(* Logix 5000 project; controller Close_Palletizing 1769-L33ERM rev 33.13; software revision 33.00; part 3 of 5 *)

ADD_ON_INSTRUCTION Generic_4PORT_IOL   (* revision 2.0 *)
// Revision note:
// 4/7/20: Changed the Input values to an input array. This makes copying the information more usable and also allows for the full Port_Process_Data_Size length.
VAR_OUTPUT
   IOL_Mode : BOOL; {access Read Only, visible}
END_VAR
VAR_IN_OUT
   PLC_Input : INT[123]; {required}
   PLC_Output : INT[87]; {required}
END_VAR
VAR_INPUT
   Port_Process_Data_Size : INT := 4; {visible}
   Port_Number : INT; {visible}
END_VAR
VAR_OUTPUT
   Vendor_ID : INT; {access Read Only, visible}
   Device_ID : DINT; {access Read Only, visible}
END_VAR
VAR_IN_OUT
   Input_Data_Array : INT[16]; {required}
   Output_Data_Array : INT[16]; {required}
END_VAR
VAR_OUTPUT
   Device_Not_Connected : BOOL; {access Read Only, visible}
   Invalid_Data : BOOL; {access Read Only, visible}
   Wrong_VID_DID : BOOL; {access Read Only, visible}
   AOI_Settings_Error : BOOL; {access Read Only, visible}
END_VAR
VAR
   Data_Size : INT; {access None}
   Offset_Address : INT; {access None}
   Offset_StatusFlgs : INT; {access None}
   Process_Offset : INT; {access None}
   RealPort_Num : INT; {access None}
   StatusFlgs_Offset : INT; {access None}
   Process_Out_Offset : INT; {access None}
END_VAR

ROUTINE Logic   (* ladder *)
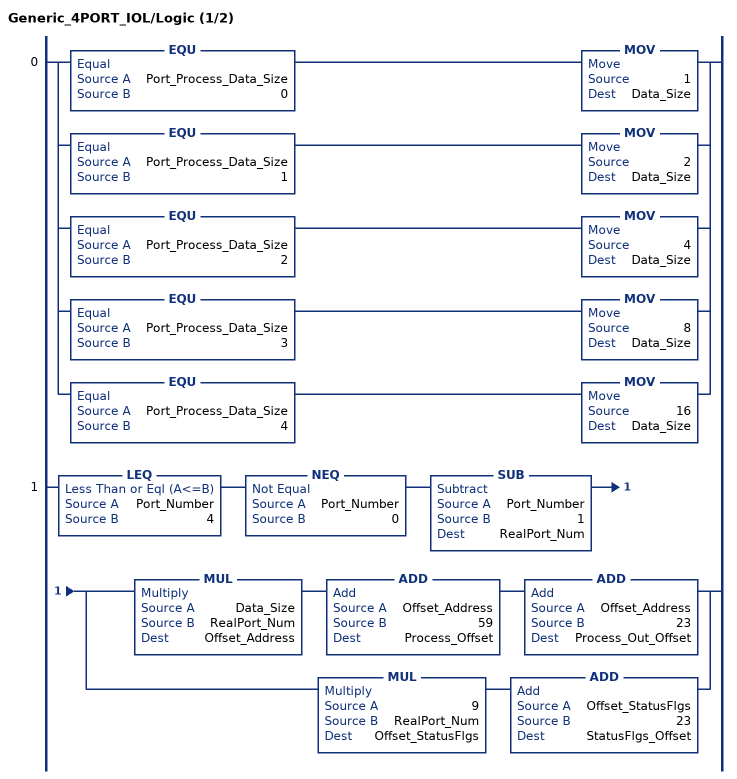
   0: [EQU(Port_Process_Data_Size,0) MOV(1,Data_Size) ,EQU(Port_Process_Data_Size,1) MOV(2,Data_Size) ,EQU(Port_Process_Data_Size,2) MOV(4,Data_Size) ,EQU(Port_Process_Data_Size,3) MOV(8,Data_Size) ,EQU(Port_Process_Data_Size,4) MOV(16,Data_Size) ];
   1: LEQ(Port_Number,4)NEQ(Port_Number,0)SUB(Port_Number,1,RealPort_Num)[MUL(Data_Size,RealPort_Num,Offset_Address) ADD(Offset_Address,59,Process_Offset) ADD(Offset_Address,23,Process_Out_Offset) ,MUL(9,RealPort_Num,Offset_StatusFlgs) ADD(Offset_StatusFlgs,23,StatusFlgs_Offset) ];
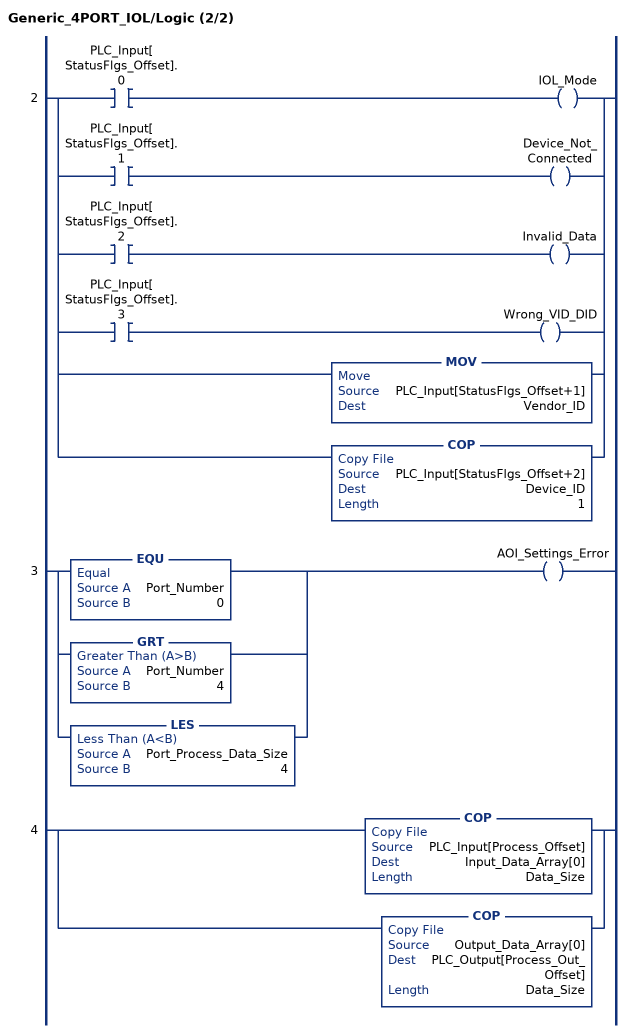
   2: [XIC(PLC_Input[StatusFlgs_Offset].0) OTE(IOL_Mode) ,XIC(PLC_Input[StatusFlgs_Offset].1) OTE(Device_Not_Connected) ,XIC(PLC_Input[StatusFlgs_Offset].2) OTE(Invalid_Data) ,XIC(PLC_Input[StatusFlgs_Offset].3) OTE(Wrong_VID_DID) ,MOV(PLC_Input[StatusFlgs_Offset+1],Vendor_ID) ,COP(PLC_Input[StatusFlgs_Offset+2],Device_ID,1) ];
   3: [EQU(Port_Number,0) ,GRT(Port_Number,4) ,LES(Port_Process_Data_Size,4) ]OTE(AOI_Settings_Error);
   4: [COP(PLC_Input[Process_Offset],Input_Data_Array[0],Data_Size) ,COP(Output_Data_Array[0],PLC_Output[Process_Out_Offset],Data_Size) ];
END_ROUTINE
END_ADD_ON_INSTRUCTION

ADD_ON_INSTRUCTION LMT_4PORT_IOL   (* revision 1.0, vendor ifm efector *)
// Cyclic Data with Diagnostics
// Revision note:
// 07/08/19 - HT
VAR_IN_OUT
   PLC_Input : INT[123]; {required}
END_VAR
VAR_INPUT
   Port_Process_Data_Size : INT := 4; {visible}
   Port_Number : INT; {visible}
END_VAR
VAR_OUTPUT
   Datastorage_Error : BOOL; {access Read Only, visible}
   Process_Data : INT; {access Read Only}
   Device_Not_Connected : BOOL; {access Read Only, visible}
   IOL_Mode : BOOL; {access Read Only, visible}
   Invalid_Data : BOOL; {access Read Only, visible}
   Media_Value : INT; {access Read Only, visible}
   Wrong_VID_DID : BOOL; {access Read Only, visible}
   Out1 : BOOL; {access Read Only, visible}
   Vendor_ID : INT; {access Read Only, visible}
   Device_ID : INT; {access Read Only, visible}
   Out2 : BOOL; {access Read Only, visible}
END_VAR
VAR
   RealPort_Num : INT; {access None}
   Offset_Address : INT; {access None}
   Process_PDI : INT; {access None}
   Process_Offset : INT; {access None}
   Offset_StatusFlgs : INT; {access None}
   StatusFlgs_Offset : INT; {access None}
   Data_Size : INT; {access None}
   Pressure_msk : INT; {access None}
END_VAR

ROUTINE Logic   (* ladder *)
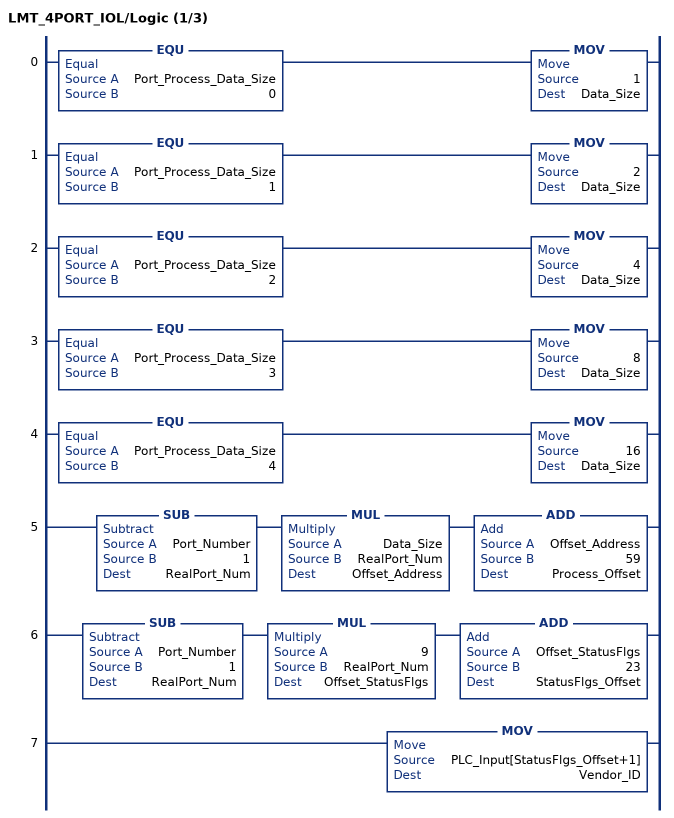
   0: EQU(Port_Process_Data_Size,0)MOV(1,Data_Size);
   1: EQU(Port_Process_Data_Size,1)MOV(2,Data_Size);
   2: EQU(Port_Process_Data_Size,2)MOV(4,Data_Size);
   3: EQU(Port_Process_Data_Size,3)MOV(8,Data_Size);
   4: EQU(Port_Process_Data_Size,4)MOV(16,Data_Size);
   5: SUB(Port_Number,1,RealPort_Num)MUL(Data_Size,RealPort_Num,Offset_Address)ADD(Offset_Address,59,Process_Offset);
   6: SUB(Port_Number,1,RealPort_Num)MUL(9,RealPort_Num,Offset_StatusFlgs)ADD(Offset_StatusFlgs,23,StatusFlgs_Offset);
   7: MOV(PLC_Input[StatusFlgs_Offset+1],Vendor_ID);
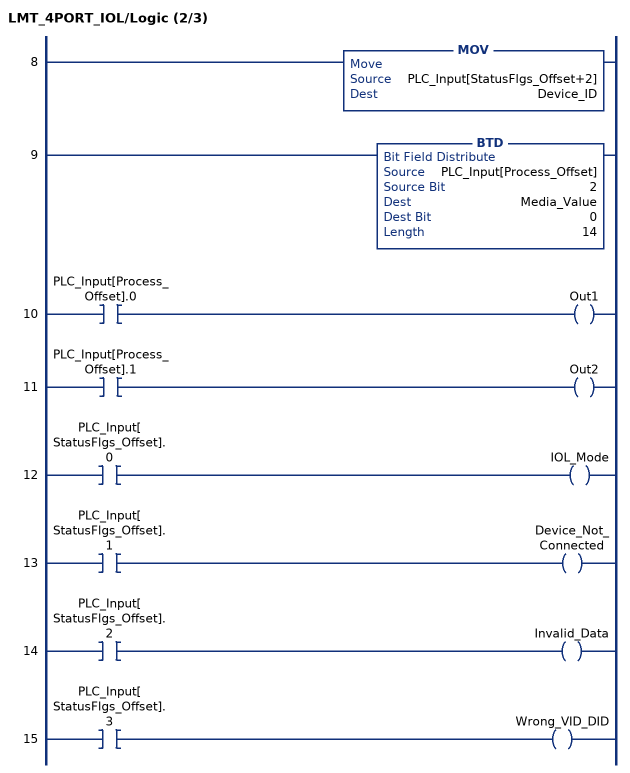
   8: MOV(PLC_Input[StatusFlgs_Offset+2],Device_ID);
   9: BTD(PLC_Input[Process_Offset],2,Media_Value,0,14);
   10: XIC(PLC_Input[Process_Offset].0)OTE(Out1);
   11: XIC(PLC_Input[Process_Offset].1)OTE(Out2);
   12: XIC(PLC_Input[StatusFlgs_Offset].0)OTE(IOL_Mode);
   13: XIC(PLC_Input[StatusFlgs_Offset].1)OTE(Device_Not_Connected);
   14: XIC(PLC_Input[StatusFlgs_Offset].2)OTE(Invalid_Data);
   15: XIC(PLC_Input[StatusFlgs_Offset].3)OTE(Wrong_VID_DID);
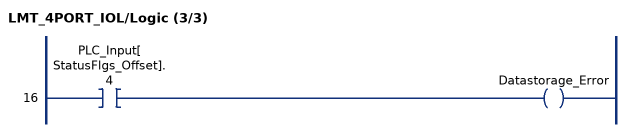
   16: XIC(PLC_Input[StatusFlgs_Offset].4)OTE(Datastorage_Error);
END_ROUTINE
END_ADD_ON_INSTRUCTION

ADD_ON_INSTRUCTION LT_4PORT_IOL   (* revision 1.0, vendor ifm efector *)
// Cyclic Data with Diagnostics
// Revision note:
// 07/08/19 - HT
VAR_IN_OUT
   PLC_Input : INT[123]; {required}
END_VAR
VAR_INPUT
   Port_Process_Data_Size : INT := 4; {visible}
   Port_Number : INT; {visible}
   Temp_Value_Gradient : REAL := 0.1; {visible}
   Level_Value_Gradient : REAL := 0.1; {visible}
END_VAR
VAR_OUTPUT
   Temperature : REAL; {access Read Only, visible}
   Datastorage_Error : BOOL; {access Read Only, visible}
   Process_Data : INT; {access Read Only}
   Device_Not_Connected : BOOL; {access Read Only, visible}
   IOL_Mode : BOOL; {access Read Only, visible}
   Invalid_Data : BOOL; {access Read Only, visible}
   Wrong_VID_DID : BOOL; {access Read Only, visible}
   Level : REAL; {access Read Only, visible}
   Out1 : BOOL; {access Read Only, visible}
   Out2 : BOOL; {access Read Only, visible}
   Vendor_ID : INT; {access Read Only, visible}
   Device_ID : INT; {access Read Only, visible}
   Out3 : BOOL; {access Read Only, visible}
   Out4 : BOOL; {access Read Only, visible}
END_VAR
VAR
   RealPort_Num : INT; {access None}
   Offset_Address : INT; {access None}
   Process_PDI : INT; {access None}
   Process_Offset : INT; {access None}
   Offset_StatusFlgs : INT; {access None}
   StatusFlgs_Offset : INT; {access None}
   Data_Size : INT; {access None}
END_VAR

ROUTINE Logic   (* ladder *)
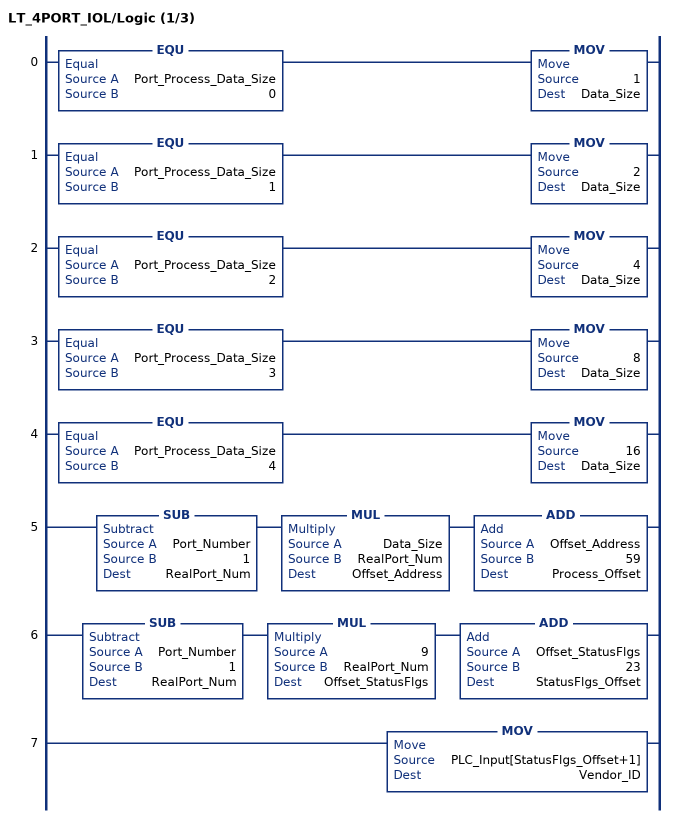
   0: EQU(Port_Process_Data_Size,0)MOV(1,Data_Size);
   1: EQU(Port_Process_Data_Size,1)MOV(2,Data_Size);
   2: EQU(Port_Process_Data_Size,2)MOV(4,Data_Size);
   3: EQU(Port_Process_Data_Size,3)MOV(8,Data_Size);
   4: EQU(Port_Process_Data_Size,4)MOV(16,Data_Size);
   5: SUB(Port_Number,1,RealPort_Num)MUL(Data_Size,RealPort_Num,Offset_Address)ADD(Offset_Address,59,Process_Offset);
   6: SUB(Port_Number,1,RealPort_Num)MUL(9,RealPort_Num,Offset_StatusFlgs)ADD(Offset_StatusFlgs,23,StatusFlgs_Offset);
   7: MOV(PLC_Input[StatusFlgs_Offset+1],Vendor_ID);
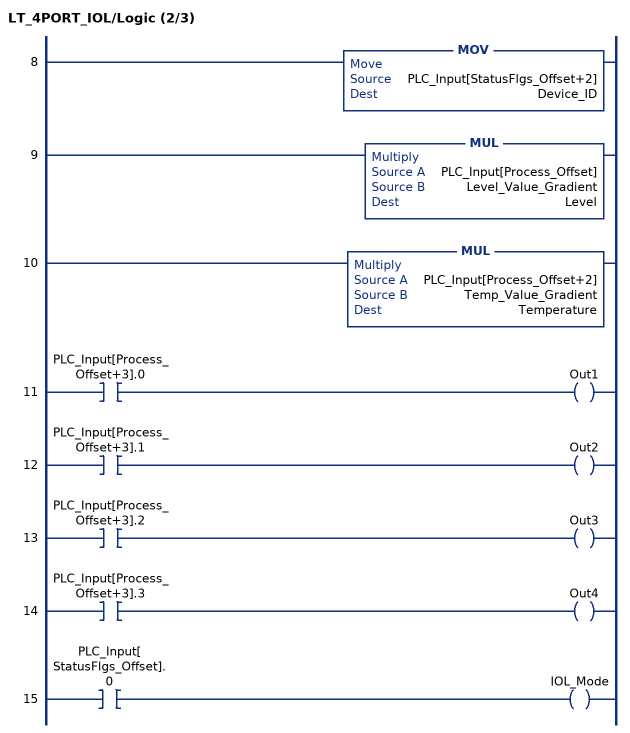
   8: MOV(PLC_Input[StatusFlgs_Offset+2],Device_ID);
   9: MUL(PLC_Input[Process_Offset],Level_Value_Gradient,Level);
   10: MUL(PLC_Input[Process_Offset+2],Temp_Value_Gradient,Temperature);
   11: XIC(PLC_Input[Process_Offset+3].0)OTE(Out1);
   12: XIC(PLC_Input[Process_Offset+3].1)OTE(Out2);
   13: XIC(PLC_Input[Process_Offset+3].2)OTE(Out3);
   14: XIC(PLC_Input[Process_Offset+3].3)OTE(Out4);
   15: XIC(PLC_Input[StatusFlgs_Offset].0)OTE(IOL_Mode);
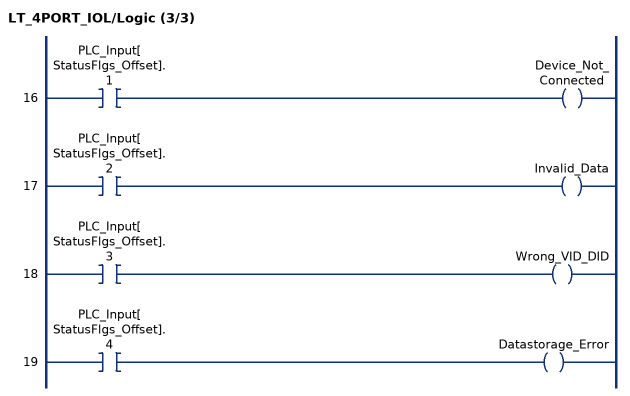
   16: XIC(PLC_Input[StatusFlgs_Offset].1)OTE(Device_Not_Connected);
   17: XIC(PLC_Input[StatusFlgs_Offset].2)OTE(Invalid_Data);
   18: XIC(PLC_Input[StatusFlgs_Offset].3)OTE(Wrong_VID_DID);
   19: XIC(PLC_Input[StatusFlgs_Offset].4)OTE(Datastorage_Error);
END_ROUTINE
END_ADD_ON_INSTRUCTION

ADD_ON_INSTRUCTION Two_AcyclicCmds_4P   (* revision 1.1 *)
// Revision note:
// 3/26/20 : On device not connected the Cmd1_DN, Cmd2_DN, Cmds_DN and Cmd_Error output bits are unlatched.
// If all Cmd Index 0, then commands are still cycled so the AL1x2x_Rdy an Cmds_DN bit still toggle on/off when the AOI is triggered.
VAR_IN_OUT
   PLC_Input : INT[123]; {required}
   PLC_Output : INT[87]; {required}
END_VAR
VAR_OUTPUT
   IOL_Mode : BOOL; {visible}
   Device_Not_Connected : BOOL; {access Read Only, visible}
   AL1x2x_Cmd_Rdy : BOOL; {visible}
   AOI_Settings_Error : BOOL; {visible}
   Cmds_Busy : BOOL; {visible}
   Cmd1_DN : BOOL; {visible}
   Cmd2_DN : BOOL; {visible}
   Cmds_DN : BOOL; {visible}
   Cmd_Errors : BOOL; {visible}
END_VAR
VAR_IN_OUT
   IOLinkMaster_Name : DINT; {required}
END_VAR
VAR_INPUT
   Port_Number : SINT; {visible}
END_VAR
VAR_OUTPUT
   Vendor_ID : INT; {access Read Only, visible}
   Device_ID : INT; {access Read Only, visible}
END_VAR
VAR_INPUT
   Cmd1_Index : INT; {visible}
   Cmd1_Subindex : INT; {visible}
   Cmd1_Rd_Wr : SINT; {visible}
   Cmd1_ByteLength : SINT; {visible}
END_VAR
VAR_IN_OUT
   Cmd1_RdWr_Buffer : SINT[32]; {required}
END_VAR
VAR_INPUT
   Cmd2_Index : INT; {visible}
   Cmd2_Subindex : INT; {visible}
   Cmd2_Rd_Wr : SINT; {visible}
   Cmd2_ByteLength : SINT; {visible}
END_VAR
VAR_IN_OUT
   Cmd2_RdWr_Buffer : SINT[32]; {required}
END_VAR
VAR_INPUT
   Cmd_Trigger : BOOL; {visible}
END_VAR
VAR_IN_OUT
   Cmd_Error_Codes : INT[2]; {required}
END_VAR
VAR_OUTPUT
   TimeOut : BOOL;
END_VAR
VAR
   Cmd1 : BOOL; {access None}
   Skip_Cmd1 : BOOL; {access None}
   Cmd1_DN_Error : BOOL; {access None}
   Cmd2 : BOOL; {access None}
   Skip_Cmd2 : BOOL; {access None}
   Cmd2_DN_Error : BOOL; {access None}
   Cmd1_Trigger : BOOL; {access None}
   Cmd2_Trigger : BOOL; {access None}
   Cmd1ReleaseTrigger : BOOL; {access None}
   Cmd2ReleaseTrigger : BOOL; {access None}
   Cmd2TriggerDelay : TIMER := (PRE := 20); {access None}
   Cmd1_PLC_OutTrigger : BOOL; {access None}
   TriggerCmdBuffer_ONS : BOOL; {access None}
   PLCTrigger : SINT; {access None}
   RealPort_Num : SINT; {access None}
   Offset_Address : INT; {access None}
   Cmd1_Busy : BOOL; {access None}
   Cmd2_Busy : BOOL; {access None}
   Offset_StatusFlgs : INT; {access None}
   StatusFlgs_Offset : INT; {access None}
   TimeOut1 : TIMER := (PRE := 6000); {access None}
   TimeOut2 : TIMER := (PRE := 6000); {access None}
   TimeOut1_Signal : BOOL; {access None}
   TimeOut2_Signal : BOOL; {access None}
   AL1x2x_Cmd_Rdy_Timer : TIMER := (PRE := 20); {access None}
   DevNotConn_Signal : BOOL; {access None}   // Signal to Latch when device is disconnected
   NoCmdSet : BOOL; {access None}
   SimCmdTimer : TIMER := (PRE := 20); {access None}
   Cmd2ReleaseTrigger_Signal : BOOL; {access None}
END_VAR

ROUTINE Logic   (* ladder *)
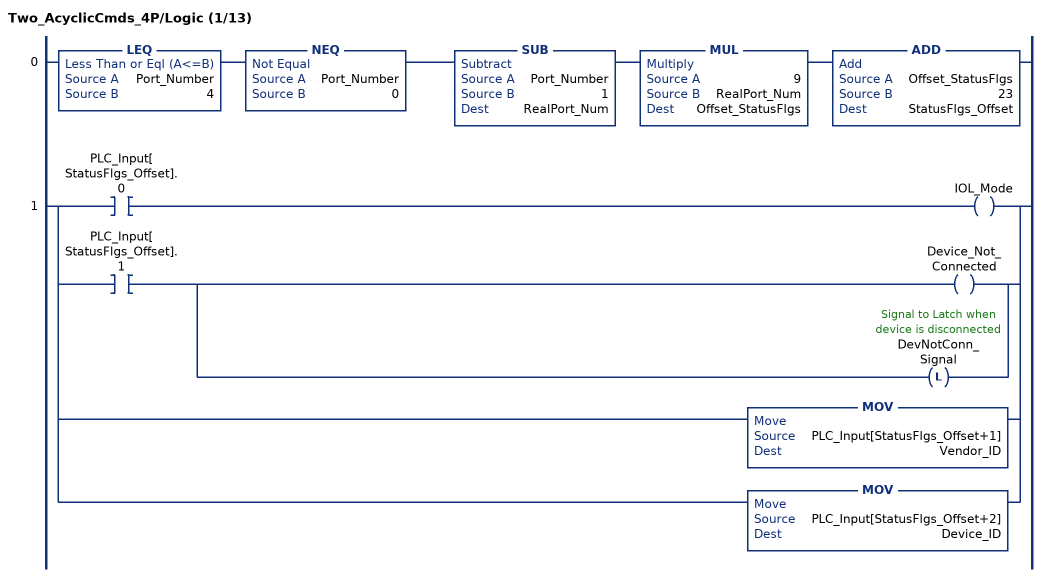
   0: LEQ(Port_Number,4)NEQ(Port_Number,0)SUB(Port_Number,1,RealPort_Num)MUL(9,RealPort_Num,Offset_StatusFlgs)ADD(Offset_StatusFlgs,23,StatusFlgs_Offset);
   1: [XIC(PLC_Input[StatusFlgs_Offset].0) OTE(IOL_Mode) ,XIC(PLC_Input[StatusFlgs_Offset].1) [OTE(Device_Not_Connected) ,OTL(DevNotConn_Signal) ] ,MOV(PLC_Input[StatusFlgs_Offset+1],Vendor_ID) ,MOV(PLC_Input[StatusFlgs_Offset+2],Device_ID) ];
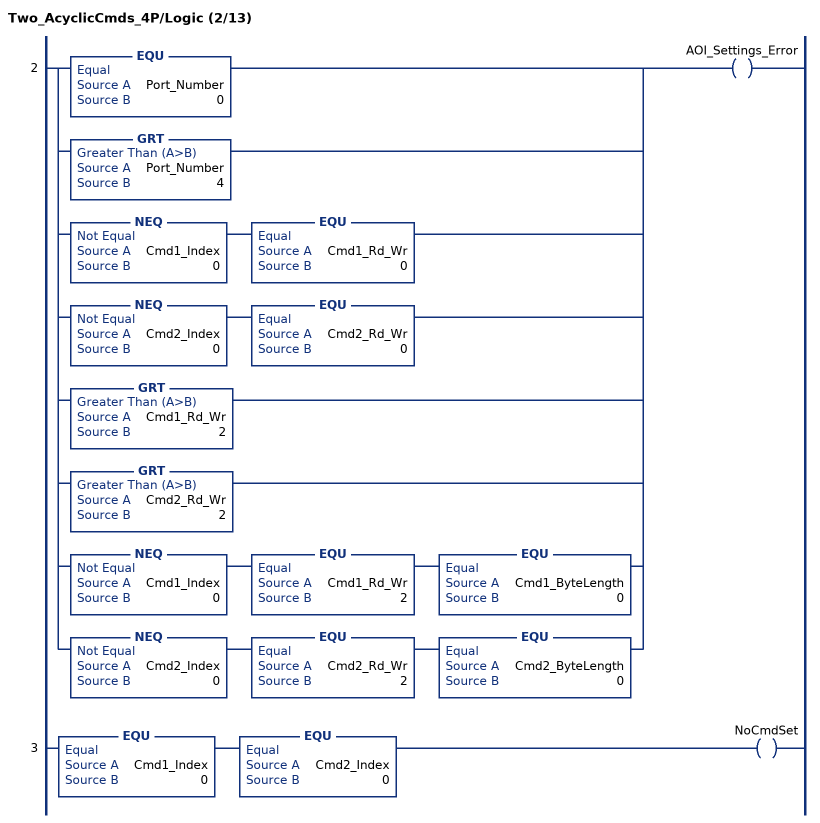
   2: [EQU(Port_Number,0) ,GRT(Port_Number,4) ,NEQ(Cmd1_Index,0) EQU(Cmd1_Rd_Wr,0) ,NEQ(Cmd2_Index,0) EQU(Cmd2_Rd_Wr,0) ,GRT(Cmd1_Rd_Wr,2) ,GRT(Cmd2_Rd_Wr,2) ,NEQ(Cmd1_Index,0) EQU(Cmd1_Rd_Wr,2) EQU(Cmd1_ByteLength,0) ,NEQ(Cmd2_Index,0) EQU(Cmd2_Rd_Wr,2) EQU(Cmd2_ByteLength,0) ]OTE(AOI_Settings_Error);
   3: EQU(Cmd1_Index,0)EQU(Cmd2_Index,0)OTE(NoCmdSet);
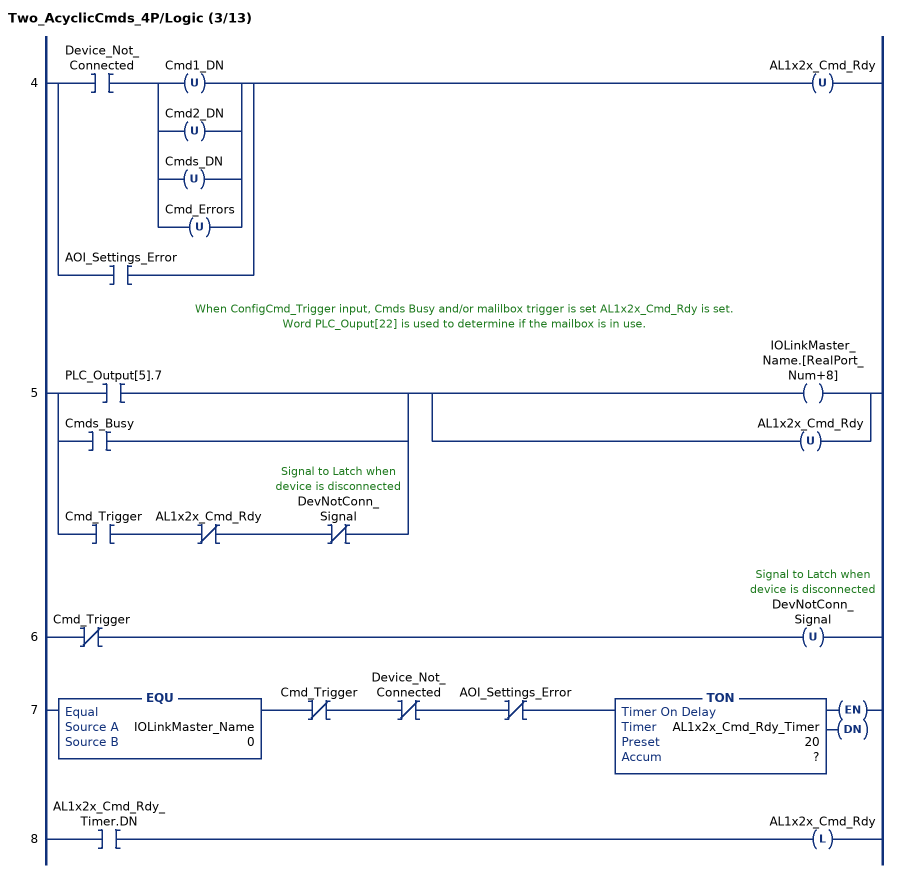
   4: [XIC(Device_Not_Connected) [OTU(Cmd1_DN) ,OTU(Cmd2_DN) ,OTU(Cmds_DN) ,OTU(Cmd_Errors) ] ,XIC(AOI_Settings_Error) ]OTU(AL1x2x_Cmd_Rdy);
   // When ConfigCmd_Trigger input, Cmds Busy and/or malilbox trigger is set AL1x2x_Cmd_Rdy is set.
   // Word PLC_Ouput[22] is used to determine if the mailbox is in use.
   5: [XIC(PLC_Output[5].7) ,XIC(Cmds_Busy) ,XIC(Cmd_Trigger) XIO(AL1x2x_Cmd_Rdy) XIO(DevNotConn_Signal) ][OTE(IOLinkMaster_Name.[RealPort_Num+8]) ,OTU(AL1x2x_Cmd_Rdy) ];
   6: XIO(Cmd_Trigger)OTU(DevNotConn_Signal);
   7: EQU(IOLinkMaster_Name,0)XIO(Cmd_Trigger)XIO(Device_Not_Connected)XIO(AOI_Settings_Error)TON(AL1x2x_Cmd_Rdy_Timer,?,?);
   8: XIC(AL1x2x_Cmd_Rdy_Timer.DN)OTL(AL1x2x_Cmd_Rdy);
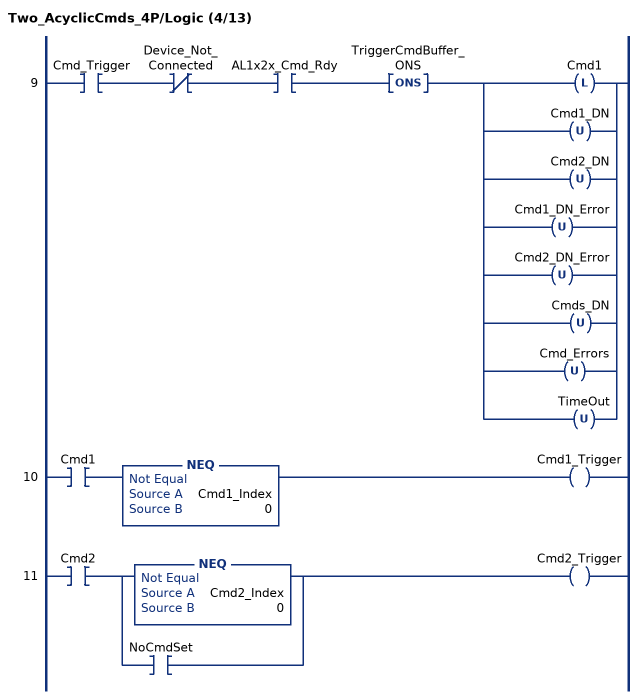
   9: XIC(Cmd_Trigger)XIO(Device_Not_Connected)XIC(AL1x2x_Cmd_Rdy)ONS(TriggerCmdBuffer_ONS)[OTL(Cmd1) ,[OTU(Cmd1_DN) ,OTU(Cmd2_DN) ,OTU(Cmd1_DN_Error) ,OTU(Cmd2_DN_Error) ,OTU(Cmds_DN) ,OTU(Cmd_Errors) ,OTU(TimeOut) ] ];
   10: XIC(Cmd1)NEQ(Cmd1_Index,0)OTE(Cmd1_Trigger);
   11: XIC(Cmd2)[NEQ(Cmd2_Index,0) ,XIC(NoCmdSet) ]OTE(Cmd2_Trigger);
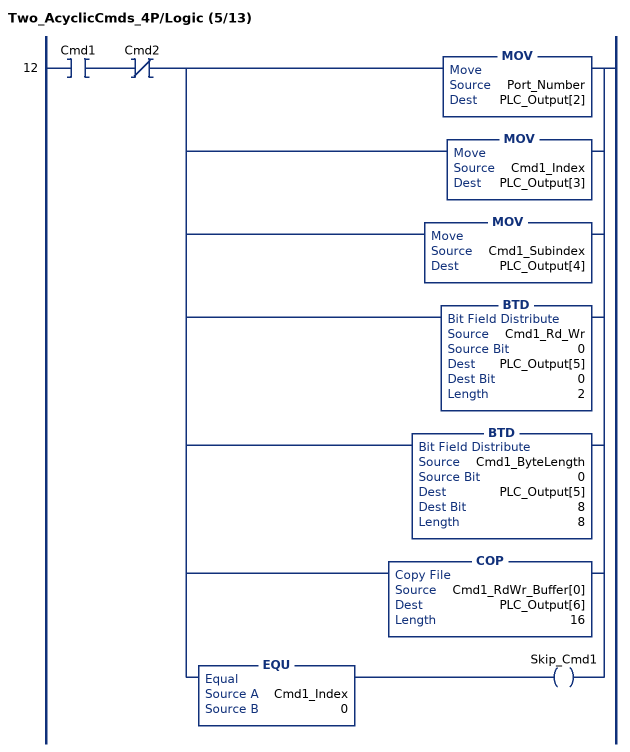
   12: XIC(Cmd1)XIO(Cmd2)[[MOV(Port_Number,PLC_Output[2]) ,MOV(Cmd1_Index,PLC_Output[3]) ,MOV(Cmd1_Subindex,PLC_Output[4]) ,BTD(Cmd1_Rd_Wr,0,PLC_Output[5],0,2) ,BTD(Cmd1_ByteLength,0,PLC_Output[5],8,8) ,COP(Cmd1_RdWr_Buffer[0],PLC_Output[6],16) ] ,EQU(Cmd1_Index,0) OTE(Skip_Cmd1) ];
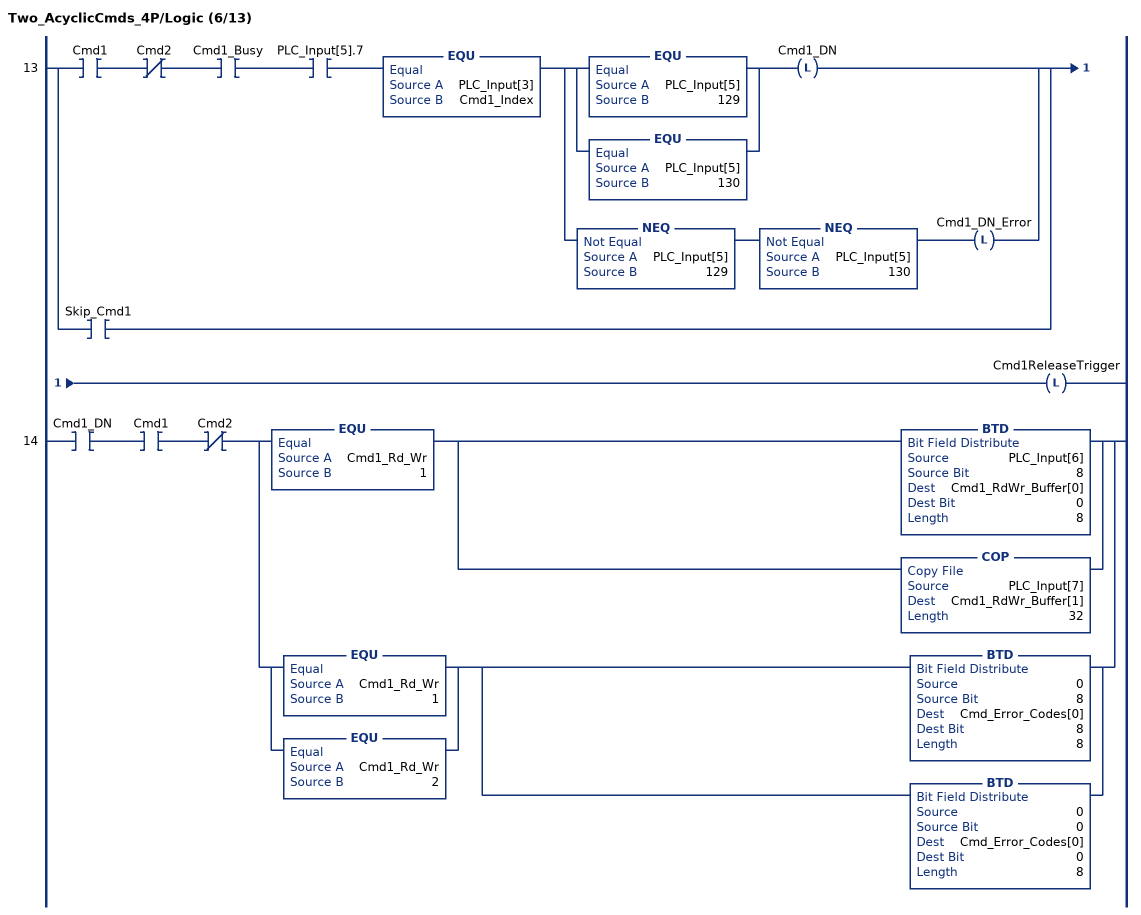
   13: [XIC(Cmd1) XIO(Cmd2) XIC(Cmd1_Busy) XIC(PLC_Input[5].7) EQU(PLC_Input[3],Cmd1_Index) [[EQU(PLC_Input[5],129) ,EQU(PLC_Input[5],130) ] OTL(Cmd1_DN) ,NEQ(PLC_Input[5],129) NEQ(PLC_Input[5],130) OTL(Cmd1_DN_Error) ] ,XIC(Skip_Cmd1) ]OTL(Cmd1ReleaseTrigger);
   14: XIC(Cmd1_DN)XIC(Cmd1)XIO(Cmd2)[EQU(Cmd1_Rd_Wr,1) [BTD(PLC_Input[6],8,Cmd1_RdWr_Buffer[0],0,8) ,COP(PLC_Input[7],Cmd1_RdWr_Buffer[1],32) ] ,[EQU(Cmd1_Rd_Wr,1) ,EQU(Cmd1_Rd_Wr,2) ] [BTD(0,8,Cmd_Error_Codes[0],8,8) ,BTD(0,0,Cmd_Error_Codes[0],0,8) ] ];
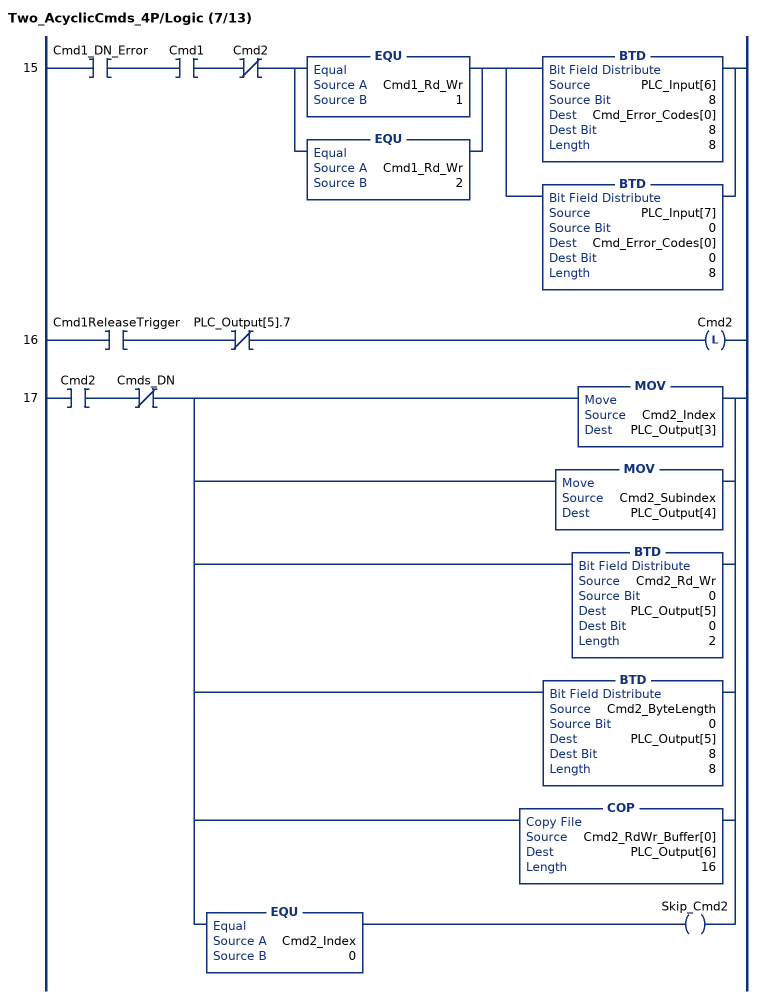
   15: XIC(Cmd1_DN_Error)XIC(Cmd1)XIO(Cmd2)[EQU(Cmd1_Rd_Wr,1) ,EQU(Cmd1_Rd_Wr,2) ][BTD(PLC_Input[6],8,Cmd_Error_Codes[0],8,8) ,BTD(PLC_Input[7],0,Cmd_Error_Codes[0],0,8) ];
   16: XIC(Cmd1ReleaseTrigger)XIO(PLC_Output[5].7)OTL(Cmd2);
   17: XIC(Cmd2)XIO(Cmds_DN)[[MOV(Cmd2_Index,PLC_Output[3]) ,MOV(Cmd2_Subindex,PLC_Output[4]) ,BTD(Cmd2_Rd_Wr,0,PLC_Output[5],0,2) ,BTD(Cmd2_ByteLength,0,PLC_Output[5],8,8) ,COP(Cmd2_RdWr_Buffer[0],PLC_Output[6],16) ] ,EQU(Cmd2_Index,0) OTE(Skip_Cmd2) ];
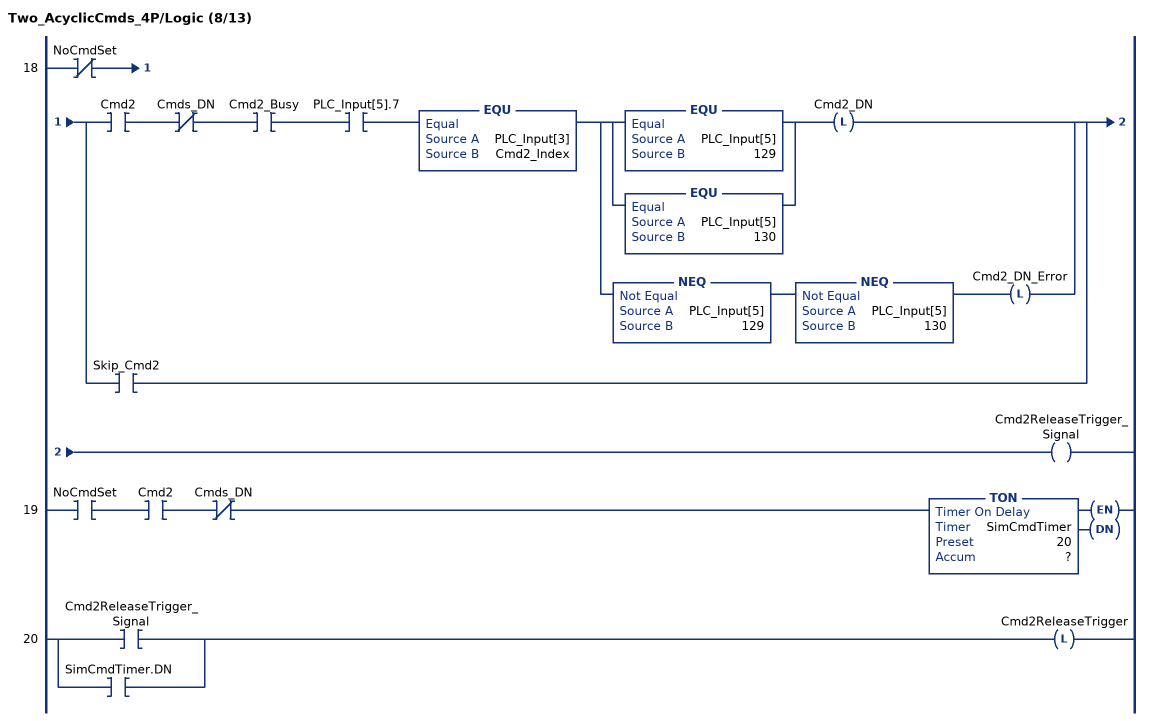
   18: XIO(NoCmdSet)[XIC(Cmd2) XIO(Cmds_DN) XIC(Cmd2_Busy) XIC(PLC_Input[5].7) EQU(PLC_Input[3],Cmd2_Index) [[EQU(PLC_Input[5],129) ,EQU(PLC_Input[5],130) ] OTL(Cmd2_DN) ,NEQ(PLC_Input[5],129) NEQ(PLC_Input[5],130) OTL(Cmd2_DN_Error) ] ,XIC(Skip_Cmd2) ]OTE(Cmd2ReleaseTrigger_Signal);
   19: XIC(NoCmdSet)XIC(Cmd2)XIO(Cmds_DN)TON(SimCmdTimer,?,?);
   20: [XIC(Cmd2ReleaseTrigger_Signal) ,XIC(SimCmdTimer.DN) ]OTL(Cmd2ReleaseTrigger);
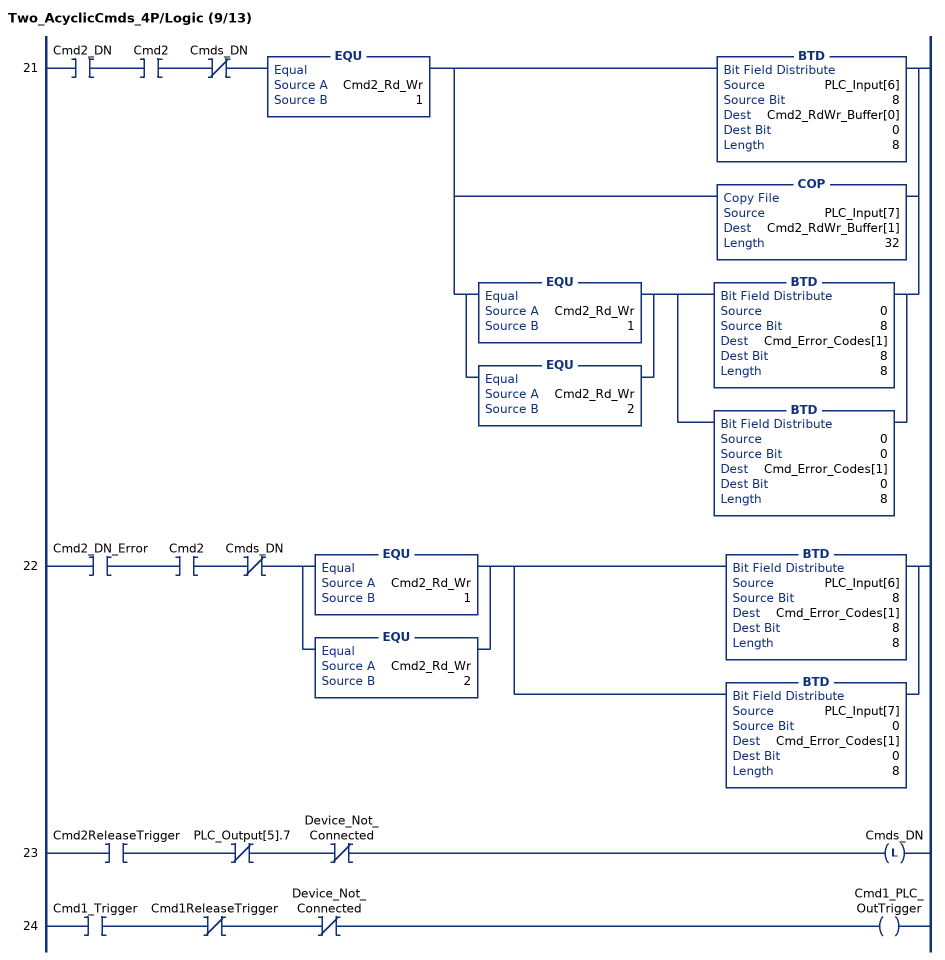
   21: XIC(Cmd2_DN)XIC(Cmd2)XIO(Cmds_DN)EQU(Cmd2_Rd_Wr,1)[[BTD(PLC_Input[6],8,Cmd2_RdWr_Buffer[0],0,8) ,COP(PLC_Input[7],Cmd2_RdWr_Buffer[1],32) ] ,[EQU(Cmd2_Rd_Wr,1) ,EQU(Cmd2_Rd_Wr,2) ] [BTD(0,8,Cmd_Error_Codes[1],8,8) ,BTD(0,0,Cmd_Error_Codes[1],0,8) ] ];
   22: XIC(Cmd2_DN_Error)XIC(Cmd2)XIO(Cmds_DN)[EQU(Cmd2_Rd_Wr,1) ,EQU(Cmd2_Rd_Wr,2) ][BTD(PLC_Input[6],8,Cmd_Error_Codes[1],8,8) ,BTD(PLC_Input[7],0,Cmd_Error_Codes[1],0,8) ];
   23: XIC(Cmd2ReleaseTrigger)XIO(PLC_Output[5].7)XIO(Device_Not_Connected)OTL(Cmds_DN);
   24: XIC(Cmd1_Trigger)XIO(Cmd1ReleaseTrigger)XIO(Device_Not_Connected)OTE(Cmd1_PLC_OutTrigger);
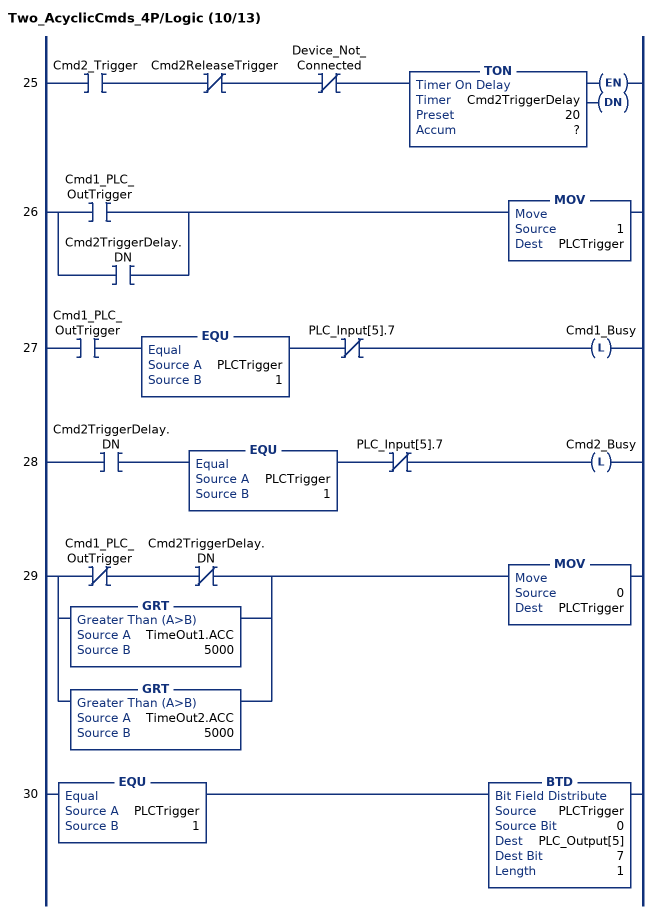
   25: XIC(Cmd2_Trigger)XIO(Cmd2ReleaseTrigger)XIO(Device_Not_Connected)TON(Cmd2TriggerDelay,?,?);
   26: [XIC(Cmd1_PLC_OutTrigger) ,XIC(Cmd2TriggerDelay.DN) ]MOV(1,PLCTrigger);
   27: XIC(Cmd1_PLC_OutTrigger)EQU(PLCTrigger,1)XIO(PLC_Input[5].7)OTL(Cmd1_Busy);
   28: XIC(Cmd2TriggerDelay.DN)EQU(PLCTrigger,1)XIO(PLC_Input[5].7)OTL(Cmd2_Busy);
   29: [XIO(Cmd1_PLC_OutTrigger) XIO(Cmd2TriggerDelay.DN) ,GRT(TimeOut1.ACC,5000) ,GRT(TimeOut2.ACC,5000) ]MOV(0,PLCTrigger);
   30: EQU(PLCTrigger,1)BTD(PLCTrigger,0,PLC_Output[5],7,1);
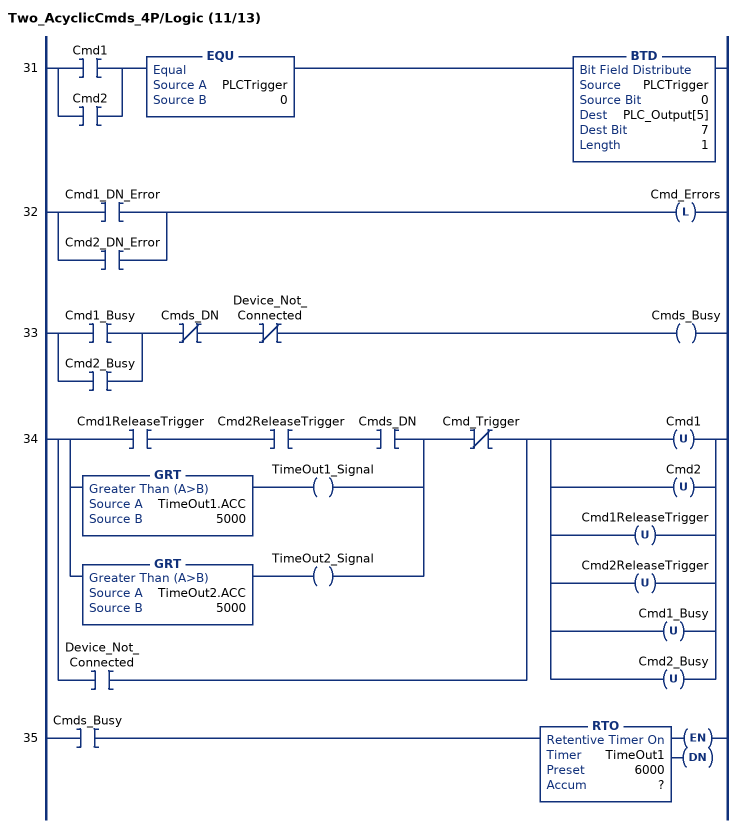
   31: [XIC(Cmd1) ,XIC(Cmd2) ]EQU(PLCTrigger,0)BTD(PLCTrigger,0,PLC_Output[5],7,1);
   32: [XIC(Cmd1_DN_Error) ,XIC(Cmd2_DN_Error) ]OTL(Cmd_Errors);
   33: [XIC(Cmd1_Busy) ,XIC(Cmd2_Busy) ]XIO(Cmds_DN)XIO(Device_Not_Connected)OTE(Cmds_Busy);
   34: [[XIC(Cmd1ReleaseTrigger) XIC(Cmd2ReleaseTrigger) XIC(Cmds_DN) ,GRT(TimeOut1.ACC,5000) OTE(TimeOut1_Signal) ,GRT(TimeOut2.ACC,5000) OTE(TimeOut2_Signal) ] XIO(Cmd_Trigger) ,XIC(Device_Not_Connected) ][OTU(Cmd1) ,OTU(Cmd2) ,OTU(Cmd1ReleaseTrigger) ,OTU(Cmd2ReleaseTrigger) ,OTU(Cmd1_Busy) ,OTU(Cmd2_Busy) ];
   35: XIC(Cmds_Busy)RTO(TimeOut1,?,?);
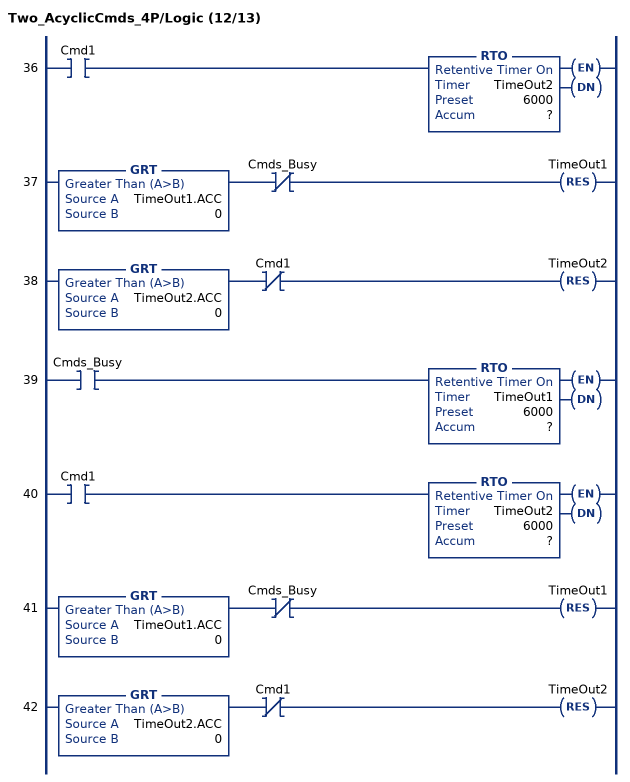
   36: XIC(Cmd1)RTO(TimeOut2,?,?);
   37: GRT(TimeOut1.ACC,0)XIO(Cmds_Busy)RES(TimeOut1);
   38: GRT(TimeOut2.ACC,0)XIO(Cmd1)RES(TimeOut2);
   39: XIC(Cmds_Busy)RTO(TimeOut1,?,?);
   40: XIC(Cmd1)RTO(TimeOut2,?,?);
   41: GRT(TimeOut1.ACC,0)XIO(Cmds_Busy)RES(TimeOut1);
   42: GRT(TimeOut2.ACC,0)XIO(Cmd1)RES(TimeOut2);
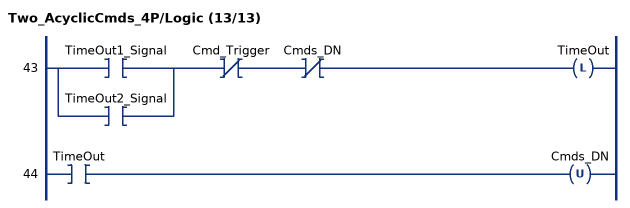
   43: [XIC(TimeOut1_Signal) ,XIC(TimeOut2_Signal) ]XIO(Cmd_Trigger)XIO(Cmds_DN)OTL(TimeOut);
   44: XIC(TimeOut)OTU(Cmds_DN);
END_ROUTINE
END_ADD_ON_INSTRUCTION
